FUNCTION ex_ARRAY_MEDIAN : REAL
VAR_INPUT
	pt: POINTER TO ARRAY[0..32000] OF REAL;
	size: UINT;
END_VAR
VAR
	i: UINT;
	stop: UINT;
END_VAR

ex_ARRAY_SORT(pt,size);
stop := SHR(size,2)-1;
IF exEVEN(UINT_TO_INT(stop)) THEN
	ex_ARRAY_MEDIAN := pt^[SHR(stop,1)];
ELSE
	i := SHR(stop,1);
	ex_ARRAY_MEDIAN := (pt^[i] + pt^[i+1]) * 0.5;
END_IF;

(* old code
stop := (size - SIZEOF(pt)) / SIZEOF(pt);
FOR i := 0 TO stop - 1 DO
	FOR m := i + 1 TO stop DO
		IF pt^[i] > pt^[m] THEN
			temp := pt^[i];
			pt^[i] := pt^[m];
			pt^[m] := temp;
		END_IF;
	END_FOR;
END_FOR;
IF even(stop) THEN
	_array_median := pt^[stop/2];
ELSE
	i := stop/2;
	_array_median := (pt^[i] + pt^[i+1])/2;
END_IF;
*)
(* revision history
hm 	3.3.2007		rev 1.1
	corrected an error, changed the statement line 14	i := TRUNC(stop/2); to i := stop/2;

hm		22. sep 2007	rev 1.2
	changed algorithm to use _array_soft for performance reasons

hm		8. oct 2007		rev 1.3
	deleted unused variables m and temp

hm		14. nov 2007	rev 1.4
	corrected a problem with size calculation

hm		16.3. 2008		rev 1.5
	changed type of input size to uint
	performance improvements
*)

END_FUNCTION

(* stored: Version 1.1.0.1, ProductVersion 3.1.4024.3
   POU ex_ARRAY_MEDIAN: Id {ea402678-cf5f-45b2-9e1e-c755bcdfea1e}, SpecialFunc None *)
